FUNCTION_BLOCK CylinderSA (* Basic Function Block Type *)
  (* Standard: 61499-2 *)
  (* Version 0.0, 2014-08-21, 4DIAC-IDE, 4DIAC-Consortium *)
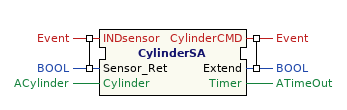
  EVENT_INPUT
    INDsensor WITH Sensor_Ret;
  END_EVENT
  EVENT_OUTPUT
    CylinderCMD WITH Extend;
  END_EVENT
  VAR_INPUT
    Sensor_Ret : BOOL; (* Input event qualifier *)
  END_VAR
  VAR_OUTPUT
    Extend : BOOL; (* Output event qualifier *)
  END_VAR
  SOCKETS
    Cylinder : ACylinder;
  END_SOCKETS
  PLUGS
    Timer : ATimeOut;
  END_PLUGS
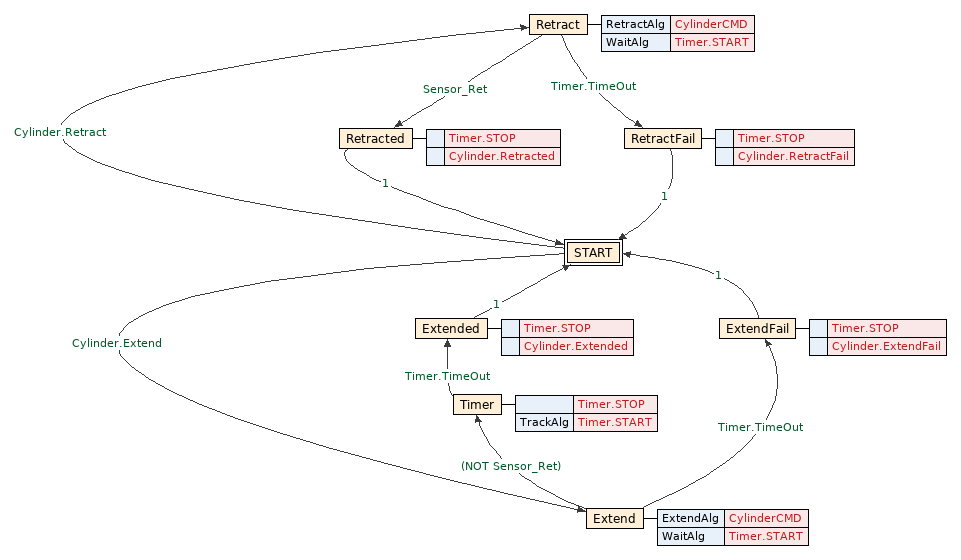
  EC_STATES
    START; (* Initial State *)
    Retract : RetractAlg -> CylinderCMD, WaitAlg -> Timer.START;
    Retracted : -> Timer.STOP, -> Cylinder.Retracted;
    Extend : ExtendAlg -> CylinderCMD, WaitAlg -> Timer.START;
    Timer : -> Timer.STOP, TrackAlg -> Timer.START;
    ExtendFail : -> Timer.STOP, -> Cylinder.ExtendFail;
    RetractFail : -> Timer.STOP, -> Cylinder.RetractFail;
    Extended : -> Timer.STOP, -> Cylinder.Extended;
  END_STATES
  EC_TRANSITIONS
    START TO Retract := Cylinder.Retract;
    START TO Extend := Cylinder.Extend;
    Timer TO Extended := Timer.TimeOut;
    Extend TO ExtendFail := Timer.TimeOut;
    Extend TO Timer := (NOT Sensor_Ret);
    RetractFail TO START := 1;
    Retracted TO START := 1;
    Extended TO START := 1;
    ExtendFail TO START := 1;
    Retract TO RetractFail := Timer.TimeOut;
    Retract TO Retracted := Sensor_Ret;
  END_TRANSITIONS
  ALGORITHM RetractAlg IN ST:
Extend:= FALSE;
  END_ALGORITHM
  ALGORITHM ExtendAlg IN ST:
Extend := TRUE;
  END_ALGORITHM
  ALGORITHM TrackAlg IN ST:
Timer.DT := T#350ms;
  END_ALGORITHM
  ALGORITHM WaitAlg IN ST: (* Time delay for sensor read *)
Timer.DT := T#5s;
  END_ALGORITHM
END_FUNCTION_BLOCK
